Staubli VAL3: session_search.pgx

program session_search(num x_nSession (dimensions=1), string& x_sSessionName[] (dimensions=1), bool& x_bFounded[] (dimensions=1))
  local num i
  local bool l_bOk
  local num l_nChar
  local num l_nSession
  local string l_sEmpty
begin
  // init
  x_bFounded=false
  x_sSessionName=""
  //
  // get the list
  //
  l_sEmpty=""
  call use:stringCopy(l_sEmpty,sSessionList)
  // get the list of session
  call saveData:getListSession(sSessionList)
  //
  // search the program from a number:
  //
  // "number+space+name"
  //
  // 01 MyPart
  // 10 YourPart
  //
  for i=0 to size(sSessionList)-1
    if sSessionList[i]!=""
      // convert the string "00 name" into a num
      toNum(sSessionList[i],l_nSession,l_bOk)
      if l_bOk and l_nSession==x_nSession
        x_sSessionName=sSessionList[i]
        x_bFounded=true
        // exit
        i=size(sSessionList)-1
      endIf
    endIf
  endFor
end
